// TIA Portal V20 export
TYPE "TypeIOLinkParamSend"
   STRUCT
      Count { ExternalAccessible := 'False'; ExternalVisible := 'False'; ExternalWritable := 'False'} : Int;
      Send { ExternalAccessible := 'False'; ExternalVisible := 'False'; ExternalWritable := 'False'} : Int;
      Info { ExternalAccessible := 'False'; ExternalVisible := 'False'; ExternalWritable := 'False'} : String[16];
      State { ExternalAccessible := 'False'; ExternalVisible := 'False'; ExternalWritable := 'False'} : Word;
   END_STRUCT;
END_TYPE
